# EPICS substitutions: heaterctrl/Db/heaterctrl.substitutions
file pid_control.db
{
pattern
{P,          PID,                              INP,                             OUT, LOPR,   HOPR, DRVL, DRVH, PREC,  KP,  KI,   KD,       SCAN}
{CstatV-AC:, PID1, CstatV-AC2:TT1A:sRdV, CstatV-AC2:EH1AB-V:cSetV,    0,  100,      0,    5,    3, 0.2,  3.,   0.,  "Passive"}
{CstatV-AC:, PID2, CstatV-AC2:TT2A:sRdV, CstatV-AC2:EH2AB-V:cSetV,    0,  100,      0,    5,    3, 0.2,  3.,   0.,  "Passive"}
{CstatV-AC:, PID3, CstatV-AC2:TT3A:sRdV, CstatV-AC2:EH3AB-V:cSetV,    0,  100,      0,    5,    3, 0.2,  3.,   0.,  "Passive"}
{CstatV-AC:, PID4, CstatV-AC2:TT4A:sRdV, CstatV-AC2:EH4AB-V:cSetV,    0,  100,      0,    5,    3, 0.2,  3.,   0.,  "Passive"}
}

file "daq6510-gen.template" { pattern
{}
{}
}

file "daq6510-chan.template" { pattern
{CHAN PID-PROC}
{01   ""}
{02   ""}
{03   ""}
{04   ""}
{05   ""}
{06   ""}
{07   ""}
{08   ""}
{09   ""}
{10   ""}
{11   "CstatV-AC:PID1.PROC"}
{12   ""}
{13   "CstatV-AC:PID2.PROC"}
{14   ""}
{15   "CstatV-AC:PID3.PROC"}
{16   "CstatV-AC:PID4.PROC"}
{17   ""}
{18   ""}
{19   ""}
{20   ""}
}

file "pid_autosave.template" { pattern
{P,          PID}
{CstatV-AC:, PID1}
{CstatV-AC:, PID2}
{CstatV-AC:, PID3}
{CstatV-AC:, PID4}
}

#file "selection.template" { pattern
#{P,     DEV}
#{CstatV-AC:DAQ6510:, PID1-Selected:RdTemp}
#}
